//structure includes axisfunctions
TYPE ST_AxFunctionsAdmin_ :
STRUCT
	Power	: MC_Power;
	Reset	: MC_Reset;
END_STRUCT
END_TYPE

(* stored: Version 1.1.0.1, ProductVersion 3.1.4024.12
   DUT ST_AxFunctionsAdmin_: Id {0e5fa7b6-9df1-4779-a9ef-6ecb4b82429b} *)
